// TIA Portal V20 export
FUNCTION "FC_Control_Manual" : Void   // FC2, LAD
{ S7_Optimized_Access := 'TRUE' }
// stored: SetENOAutomatically false
BEGIN

REGION Network 1: Solenoide Salida Cilindro 1
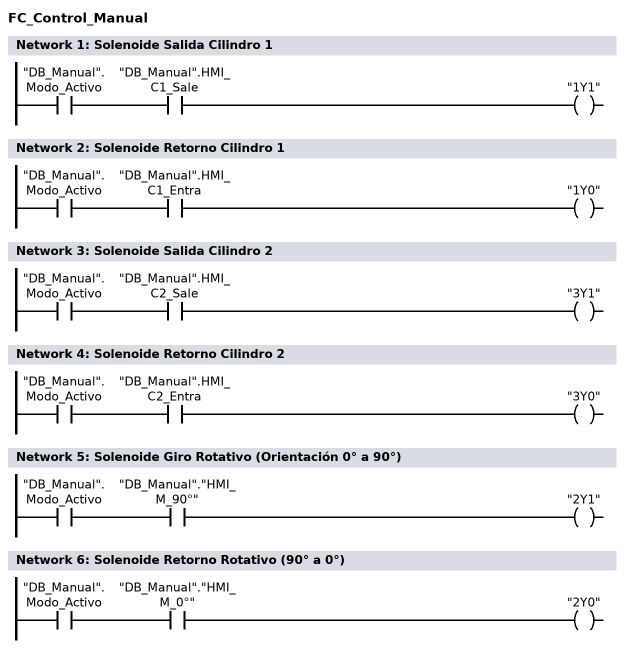
   RUNG wire#powerrail
      Contact( "DB_Manual".Modo_Activo )
      Contact( "DB_Manual".HMI_C1_Sale )
      Coil( "1Y1" )
   END_RUNG
   // the same network as SCL:
   "1Y1" := "DB_Manual".Modo_Activo AND "DB_Manual".HMI_C1_Sale;
END_REGION

REGION Network 2: Solenoide Retorno Cilindro 1
   RUNG wire#powerrail
      Contact( "DB_Manual".Modo_Activo )
      Contact( "DB_Manual".HMI_C1_Entra )
      Coil( "1Y0" )
   END_RUNG
   // the same network as SCL:
   "1Y0" := "DB_Manual".Modo_Activo AND "DB_Manual".HMI_C1_Entra;
END_REGION

REGION Network 3: Solenoide Salida Cilindro 2
   RUNG wire#powerrail
      Contact( "DB_Manual".Modo_Activo )
      Contact( "DB_Manual".HMI_C2_Sale )
      Coil( "3Y1" )
   END_RUNG
   // the same network as SCL:
   "3Y1" := "DB_Manual".Modo_Activo AND "DB_Manual".HMI_C2_Sale;
END_REGION

REGION Network 4: Solenoide Retorno Cilindro 2
   RUNG wire#powerrail
      Contact( "DB_Manual".Modo_Activo )
      Contact( "DB_Manual".HMI_C2_Entra )
      Coil( "3Y0" )
   END_RUNG
   // the same network as SCL:
   "3Y0" := "DB_Manual".Modo_Activo AND "DB_Manual".HMI_C2_Entra;
END_REGION

REGION Network 5: Solenoide Giro Rotativo (Orientación 0° a 90°)
   RUNG wire#powerrail
      Contact( "DB_Manual".Modo_Activo )
      Contact( "DB_Manual"."HMI_M_90°" )
      Coil( "2Y1" )
   END_RUNG
   // the same network as SCL:
   "2Y1" := "DB_Manual".Modo_Activo AND "DB_Manual"."HMI_M_90°";
END_REGION

REGION Network 6: Solenoide Retorno Rotativo (90° a 0°)
   RUNG wire#powerrail
      Contact( "DB_Manual".Modo_Activo )
      Contact( "DB_Manual"."HMI_M_0°" )
      Coil( "2Y0" )
   END_RUNG
   // the same network as SCL:
   "2Y0" := "DB_Manual".Modo_Activo AND "DB_Manual"."HMI_M_0°";
END_REGION
END_FUNCTION
